# EPICS substitutions: ioc/bsread_test.subs
file bsread_test.template {
	pattern{P} {BSREAD-TEST}
}
